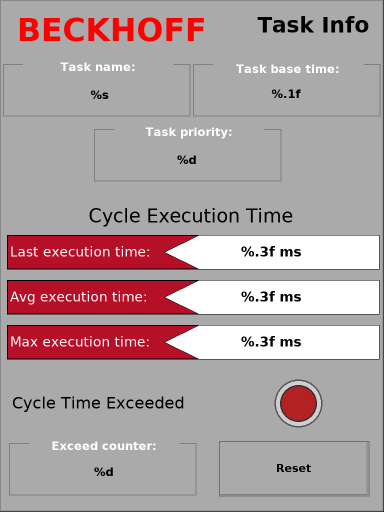
VISUALIZATION PH_TaskInfo  // 384x512
VAR_IN_OUT
	fbTaskInfo	:FB_TaskInfo;
END_VAR
    Rectangle (0,0 384x512)
    Label (9,10 206x40), "BECKHOFF"
    Label (242,10 143x30), "Task Info"
    RoundedRectangle (3,64 187x52)
    Rectangle (23,52 150x30), "Task name:"
    RoundedRectangle (193,64 187x52)
    Rectangle (213,54 150x30), "Task base time:"
    RoundedRectangle (7,235 205x34), "Last execution time:"
    Polygon (164,252) (199,235) (379,235) (379,269) (199,269), "%.3f ms", text variable: fbTaskInfo.rLastExecTime
    RoundedRectangle (94,129 187x52)
    Rectangle (114,117 150x30), "Task priority:"
    Label (-1,201 384x30), "Cycle Execution Time"
    RoundedRectangle (7,280 205x34), "Avg execution time:"
    Polygon (164,297) (199,280) (379,280) (379,314) (199,314), "%.3f ms", text variable: fbTaskInfo.rAverageCycleTime
    RoundedRectangle (7,325 205x34), "Max execution time:"
    Polygon (164,342) (199,325) (379,325) (379,359) (199,359), "%.3f ms", text variable: fbTaskInfo.rMaxExecTime
    Label (9,388 251x30), "Cycle Time Exceeded"
    Lamp1 (271,376 55x55), variable: fbTaskInfo.bCycleTimeExceeded, style: Lamp-Lamp1-Red
    RoundedRectangle (9,443 187x52)
    Rectangle (29,431 150x30), "Exceed counter:"
    Button (219,441 150x55), "Reset"
        tap fbTaskInfo.bResetVisu
    Rectangle (25,80 150x30), "%s", text variable: fbTaskInfo.sTaskName
    Rectangle (211,79 150x30), "%.1f", text variable: fbTaskInfo.rCycleTime
    Rectangle (112,145 150x30), "%d", text variable: fbTaskInfo.uiPriority
    Rectangle (29,457 150x30), "%d", text variable: fbTaskInfo.udiCountExceedCycle
END_VISUALIZATION

(* stored: Version 1.1.0.1, ProductVersion 3.1.4024.5
   Visu PH_TaskInfo: Id {6aa8c01d-c79f-47af-b844-018f75c0812d} *)
